TYPE DUT_SimMotorStates :
(
	IDLE := 0, 
	CHECK,
	MOVING
);
END_TYPE

(* stored: Version 1.1.0.1, ProductVersion 3.1.4024.2
   DUT DUT_SimMotorStates: Id {6a981ff5-0d13-4f8b-97d8-6e15ecc8935f} *)
